FUNCTION_BLOCK FB_ADS
VAR_INPUT
END_VAR
VAR_OUTPUT
END_VAR
VAR
     fbLogger : FB_LogMessage := (eSubsystem:=E_SubSystem.FIELDBUS);
    tErrorPresent : R_TRIG;
END_VAR

END_FUNCTION_BLOCK

(* stored: Version 1.1.0.1
   POU FB_ADS: Id {ab53a300-a8c7-4757-a8eb-e10b4abda9ef}, SpecialFunc None *)
